// Mitsubishi GX Works2 project: b05   PLC: Q02/Q02H

PROGRAM MAIN
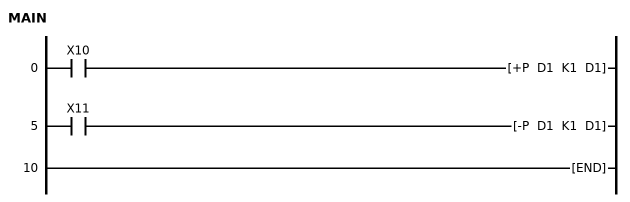
0     LD      X10
      +P      D1 K1 D1
5     LD      X11
      -P      D1 K1 D1
10    END
END_PROGRAM
